            movement171ActiveLeft : Bool;   // Movement Active
            movement171ActiveRight : Bool;   // Movement Active
            movement172ActiveLeft : Bool;   // Movement Active
            movement172ActiveRight : Bool;   // Movement Active
            movement173ActiveLeft : Bool;   // Movement Active
            movement173ActiveRight : Bool;   // Movement Active
            movement174ActiveLeft : Bool;   // Movement Active
            movement174ActiveRight : Bool;   // Movement Active
            movement175ActiveLeft : Bool;   // Movement Active
            movement175ActiveRight : Bool;   // Movement Active
            movement176ActiveLeft : Bool;   // Movement Active
            movement176ActiveRight : Bool;   // Movement Active
            movement177ActiveLeft : Bool;   // Movement Active
            movement177ActiveRight : Bool;   // Movement Active
            movement178ActiveLeft : Bool;   // Movement Active
            movement178ActiveRight : Bool;   // Movement Active
            movement179ActiveLeft : Bool;   // Movement Active
            movement179ActiveRight : Bool;   // Movement Active
            movement180ActiveLeft : Bool;   // Movement Active
            movement180ActiveRight : Bool;   // Movement Active
            movement181ActiveLeft : Bool;   // Movement Active
            movement181ActiveRight : Bool;   // Movement Active
            movement182ActiveLeft : Bool;   // Movement Active
            movement182ActiveRight : Bool;   // Movement Active
            movement183ActiveLeft : Bool;   // Movement Active
            movement183ActiveRight : Bool;   // Movement Active
            movement184ActiveLeft : Bool;   // Movement Active
            movement184ActiveRight : Bool;   // Movement Active
            movement185ActiveLeft : Bool;   // Movement Active
            movement185ActiveRight : Bool;   // Movement Active
            movement186ActiveLeft : Bool;   // Movement Active
            movement186ActiveRight : Bool;   // Movement Active
            movement187ActiveLeft : Bool;   // Movement Active
            movement187ActiveRight : Bool;   // Movement Active
            movement188ActiveLeft : Bool;   // Movement Active
            movement188ActiveRight : Bool;   // Movement Active
            movement189ActiveLeft : Bool;   // Movement Active
            movement189ActiveRight : Bool;   // Movement Active
            movement190ActiveLeft : Bool;   // Movement Active
            movement190ActiveRight : Bool;   // Movement Active
            movement191ActiveLeft : Bool;   // Movement Active
            movement191ActiveRight : Bool;   // Movement Active
            movement192ActiveLeft : Bool;   // Movement Active
            movement192ActiveRight : Bool;   // Movement Active
            movement193ActiveLeft : Bool;   // Movement Active
            movement193ActiveRight : Bool;   // Movement Active
            movement194ActiveLeft : Bool;   // Movement Active
            movement194ActiveRight : Bool;   // Movement Active
            movement195ActiveLeft : Bool;   // Movement Active
            movement195ActiveRight : Bool;   // Movement Active
            movement196ActiveLeft : Bool;   // Movement Active
            movement196ActiveRight : Bool;   // Movement Active
            movement197ActiveLeft : Bool;   // Movement Active
            movement197ActiveRight : Bool;   // Movement Active
            movement198ActiveLeft : Bool;   // Movement Active
            movement198ActiveRight : Bool;   // Movement Active
            movement199ActiveLeft : Bool;   // Movement Active
            movement199ActiveRight : Bool;   // Movement Active
            movement200ActiveLeft : Bool;   // Movement Active
            movement200ActiveRight : Bool;   // Movement Active
            movement201ActiveLeft : Bool;   // Movement Active
            movement201ActiveRight : Bool;   // Movement Active
            movement202ActiveLeft : Bool;   // Movement Active
            movement202ActiveRight : Bool;   // Movement Active
            movement203ActiveLeft : Bool;   // Movement Active
            movement203ActiveRight : Bool;   // Movement Active
            movement204ActiveLeft : Bool;   // Movement Active
            movement204ActiveRight : Bool;   // Movement Active
            movement205ActiveLeft : Bool;   // Movement Active
            movement205ActiveRight : Bool;   // Movement Active
            movement206ActiveLeft : Bool;   // Movement Active
            movement206ActiveRight : Bool;   // Movement Active
            movement207ActiveLeft : Bool;   // Movement Active
            movement207ActiveRight : Bool;   // Movement Active
            movement208ActiveLeft : Bool;   // Movement Active
            movement208ActiveRight : Bool;   // Movement Active
            movement209ActiveLeft : Bool;   // Movement Active
            movement209ActiveRight : Bool;   // Movement Active
            movement210ActiveLeft : Bool;   // Movement Active
            movement210ActiveRight : Bool;   // Movement Active
            movement211ActiveLeft : Bool;   // Movement Active
            movement211ActiveRight : Bool;   // Movement Active
            movement212ActiveLeft : Bool;   // Movement Active
            movement212ActiveRight : Bool;   // Movement Active
            movement213ActiveLeft : Bool;   // Movement Active
            movement213ActiveRight : Bool;   // Movement Active
            movement214ActiveLeft : Bool;   // Movement Active
            movement214ActiveRight : Bool;   // Movement Active
            movement215ActiveLeft : Bool;   // Movement Active
            movement215ActiveRight : Bool;   // Movement Active
            movement216ActiveLeft : Bool;   // Movement Active
            movement216ActiveRight : Bool;   // Movement Active
            movement217ActiveLeft : Bool;   // Movement Active
            movement217ActiveRight : Bool;   // Movement Active
            movement218ActiveLeft : Bool;   // Movement Active
            movement218ActiveRight : Bool;   // Movement Active
            movement219ActiveLeft : Bool;   // Movement Active
            movement219ActiveRight : Bool;   // Movement Active
            movement220ActiveLeft : Bool;   // Movement Active
            movement220ActiveRight : Bool;   // Movement Active
            movement221ActiveLeft : Bool;   // Movement Active
            movement221ActiveRight : Bool;   // Movement Active
            movement222ActiveLeft : Bool;   // Movement Active
            movement222ActiveRight : Bool;   // Movement Active
            movement223ActiveLeft : Bool;   // Movement Active
            movement223ActiveRight : Bool;   // Movement Active
            movement224ActiveLeft : Bool;   // Movement Active
            movement224ActiveRight : Bool;   // Movement Active
            movement225ActiveLeft : Bool;   // Movement Active
            movement225ActiveRight : Bool;   // Movement Active
            movement226ActiveLeft : Bool;   // Movement Active
            movement226ActiveRight : Bool;   // Movement Active
            movement227ActiveLeft : Bool;   // Movement Active
            movement227ActiveRight : Bool;   // Movement Active
            movement228ActiveLeft : Bool;   // Movement Active
            movement228ActiveRight : Bool;   // Movement Active
            movement229ActiveLeft : Bool;   // Movement Active
            movement229ActiveRight : Bool;   // Movement Active
            movement230ActiveLeft : Bool;   // Movement Active
            movement230ActiveRight : Bool;   // Movement Active
            movement231ActiveLeft : Bool;   // Movement Active
            movement231ActiveRight : Bool;   // Movement Active
            movement232ActiveLeft : Bool;   // Movement Active
            movement232ActiveRight : Bool;   // Movement Active
            movement233ActiveLeft : Bool;   // Movement Active
            movement233ActiveRight : Bool;   // Movement Active
            movement234ActiveLeft : Bool;   // Movement Active
            movement234ActiveRight : Bool;   // Movement Active
            movement235ActiveLeft : Bool;   // Movement Active
            movement235ActiveRight : Bool;   // Movement Active
            movement236ActiveLeft : Bool;   // Movement Active
            movement236ActiveRight : Bool;   // Movement Active
            movement237ActiveLeft : Bool;   // Movement Active
            movement237ActiveRight : Bool;   // Movement Active
            movement238ActiveLeft : Bool;   // Movement Active
            movement238ActiveRight : Bool;   // Movement Active
            movement239ActiveLeft : Bool;   // Movement Active
            movement239ActiveRight : Bool;   // Movement Active
            movement240ActiveLeft : Bool;   // Movement Active
            movement240ActiveRight : Bool;   // Movement Active
            movement241ActiveLeft : Bool;   // Movement Active
            movement241ActiveRight : Bool;   // Movement Active
            movement242ActiveLeft : Bool;   // Movement Active
            movement242ActiveRight : Bool;   // Movement Active
            movement243ActiveLeft : Bool;   // Movement Active
            movement243ActiveRight : Bool;   // Movement Active
            movement244ActiveLeft : Bool;   // Movement Active
            movement244ActiveRight : Bool;   // Movement Active
            movement245ActiveLeft : Bool;   // Movement Active
            movement245ActiveRight : Bool;   // Movement Active
            movement246ActiveLeft : Bool;   // Movement Active
            movement246ActiveRight : Bool;   // Movement Active
            movement247ActiveLeft : Bool;   // Movement Active
            movement247ActiveRight : Bool;   // Movement Active
            movement248ActiveLeft : Bool;   // Movement Active
            movement248ActiveRight : Bool;   // Movement Active
            movement249ActiveLeft : Bool;   // Movement Active
            movement249ActiveRight : Bool;   // Movement Active
            movement250ActiveLeft : Bool;   // Movement Active
            movement250ActiveRight : Bool;   // Movement Active
            movement251ActiveLeft : Bool;   // Movement Active
            movement251ActiveRight : Bool;   // Movement Active
            movement252ActiveLeft : Bool;   // Movement Active
            movement252ActiveRight : Bool;   // Movement Active
            movement253ActiveLeft : Bool;   // Movement Active
            movement253ActiveRight : Bool;   // Movement Active
            movement254ActiveLeft : Bool;   // Movement Active
            movement254ActiveRight : Bool;   // Movement Active
            movement255ActiveLeft : Bool;   // Movement Active
            movement255ActiveRight : Bool;   // Movement Active
            movement256ActiveLeft : Bool;   // Movement Active
            movement256ActiveRight : Bool;   // Movement Active
         END_STRUCT;
      END_STRUCT;
   END_VAR
BEGIN
END_DATA_BLOCK
